(* IEC 61131-3 sources: moqui-plc/simatic-ax/src/moqui/framework/src/main/org/moqui/context, 9 files *)

(* ---- LogCmd.st ---- *)
TYPE LogCmd : (
    Idle, (* Waiting for commands *)
    Push, (* Inserting a new log entry *)
	IncrementLast, (* Update the last log entry *)
	Peek, (* Read a log entry without removing it *)
	Pop, (* It actually removes the appended log entries *)
    Clear (* Complete buffer reset *)
); END_TYPE

(* ---- LogEvent.st ---- *)
TYPE LogEvent : STRUCT
	(* Unique identifier for the log event *)
    logEventId : STRING;
    loggerName : STRING;
	marker : LogMarker;
    level : LogLevel;
    logEventDate : DATE_AND_TIME;
	source : STRING;
	payloadType : LogPayloadType;
    payload : LogPayload;
	(* contextData: STRING; *)
	(* Number of times this log event was repeated, for compression *)
    repeatCount : UINT;
END_STRUCT; END_TYPE

(* ---- LogLevel.st ---- *)
TYPE LogLevel : (
	Trace,
	Debug,
	Info,
	Warn,
	Error,
	Fatal,
	All,
	Off
); END_TYPE

(* ---- LogMarker.st ---- *)
TYPE LogMarker : (
	Diagnostics,
	Lifecycle,
	Integration,
	Health,
	Telemetry,
	AuditLog,
	Kpi,
	Measurement
); END_TYPE

(* ---- LogPayload.st ---- *)
TYPE LogPayload : STRUCT
	message : STRING;
    enumValue : UINT;
    numericValue : LREAL;
END_STRUCT; END_TYPE

(* ---- LogPayloadType.st ---- *)
TYPE LogPayloadType : (
    Text,
	Numeric,
	Enum
); END_TYPE

(* ---- LogSource.st ---- *)
TYPE LogSource : STRUCT
	(* Reference to log ring buffer *)
    logRef : REF_TO LogRingBuffer;
	lastLogSize : UINT;
	lastHead : UINT := UINT#1;
	lastTail : UINT := UINT#1;
	lastOverflowCount : UDINT;
END_STRUCT; END_TYPE

(* ---- LoggerFacade.st ---- *)
(*
 * Logger with local circular buffer and duplicate suppression.
 * Designed for central orchestration by a global LogAppender.
 *)
FUNCTION_BLOCK LoggerFacade
	VAR_EXTERNAL CONSTANT
		defaultLogLevel : LogLevel;
		defaultLogSuppressDuration : TIME;
		defaultLogSuppressDuplicates : BOOL;
		LOG_SOURCE_LIST_MAX_SIZE : UINT;
	END_VAR
	VAR_EXTERNAL
		logSourceList : ARRAY[1..LOG_SOURCE_LIST_MAX_SIZE] OF LogSource;
		logSourceListSize : UINT;
	END_VAR
	(* Log event data *)
	VAR_INPUT
		enable : BOOL;
		logEventId : STRING := '';
		loggerName : STRING;
		level : LogLevel := defaultLogLevel;
		marker : LogMarker := LogMarker#Diagnostics;
		source : STRING;
		payloadType : LogPayloadType := LogPayloadType#Text;
		message : STRING;
		enumValue : UINT;
		numericValue : LREAL;
	END_VAR
	(* Configuration parameters *)
	VAR_INPUT
		suppressDuplicates : BOOL := defaultLogSuppressDuplicates;
		suppressDuration : TIME := defaultLogSuppressDuration;
	END_VAR
	VAR_OUTPUT
		done : BOOL;
		error : BOOL;
	END_VAR
	VAR
		(* Local log ring buffer *)
		logBuffer : LogRingBuffer;
		init : BOOL := FALSE;
		isDuplicate : BOOL;
		now : DATE_AND_TIME;
		lastLogEvent : LogEvent;
		(* Log event ID generator *)
		eventSequence : UDINT := UDINT#0;
	END_VAR

	(* Register once into the log appender source list *)
	IF NOT init THEN
		IF logSourceListSize < LOG_SOURCE_LIST_MAX_SIZE THEN
			logSourceListSize := logSourceListSize + UINT#1;
			logSourceList[logSourceListSize].logRef := REF(logBuffer);
		ELSE
			error := TRUE;
		END_IF;
		init := TRUE;
	END_IF;

	IF NOT enable THEN
		done := FALSE;
		RETURN;
	END_IF;

	now := nowTimestamp();
	isDuplicate := FALSE;

	(* Compression logic (duplicate suppression) *)
	IF suppressDuplicates AND (payloadType = lastLogEvent.payloadType)
			AND (loggerName = lastLogEvent.loggerName)
			AND (source = lastLogEvent.source) THEN
		CASE payloadType OF
			LogPayloadType#Text: isDuplicate := (message = lastLogEvent.payload.message);
			LogPayloadType#Enum: isDuplicate := (enumValue = lastLogEvent.payload.enumValue);
			LogPayloadType#Numeric: isDuplicate := (numericValue = lastLogEvent.payload.numericValue);
		END_CASE;
	END_IF;

	IF isDuplicate AND ((now - lastLogEvent.logEventDate) < suppressDuration) THEN
		(* Increment repeat counter instead of storing new entry *)
		logBuffer.cmd := LogCmd#IncrementLast;
	ELSE
		(* Prepare the new log event entry *)
		IF logEventId = '' THEN
			eventSequence := eventSequence + UDINT#1;
			lastLogEvent.logEventId := loggerName;
		ELSE
			lastLogEvent.logEventId := logEventId;
		END_IF;

		lastLogEvent.loggerName := loggerName;
		lastLogEvent.level := level;
		lastLogEvent.marker := marker;
		lastLogEvent.logEventDate := now;
		lastLogEvent.source := source;
		lastLogEvent.payloadType := payloadType;
		lastLogEvent.repeatCount := UINT#1;

		CASE payloadType OF
			LogPayloadType#Text: lastLogEvent.payload.message := message;
			LogPayloadType#Enum: lastLogEvent.payload.enumValue := enumValue;
			LogPayloadType#Numeric: lastLogEvent.payload.numericValue := numericValue;
		END_CASE;

		(* Append the new log event *)
		logBuffer.logEntry := lastLogEvent;
		logBuffer.cmd := LogCmd#Push;
	END_IF;

	(* Execute local buffer operation *)
	logBuffer();
	logBuffer.cmd := LogCmd#Idle;

	done := logBuffer.done;
	error := error OR logBuffer.error;
END_FUNCTION_BLOCK

(* ---- LogRingBuffer.st ---- *)
FUNCTION_BLOCK LogRingBuffer
	VAR_EXTERNAL CONSTANT
	    LOG_MAX_SIZE : UINT;
	END_VAR
	VAR_INPUT
	    cmd : LogCmd := LogCmd#Idle;
	    logEntry : LogEvent;
	END_VAR
	VAR_OUTPUT
	    done, error, isFull, isEmpty : BOOL;
	    head : UINT := UINT#1;
	    tail : UINT := UINT#1;
	    (* Peek/Pop result: set on LogCmd#Peek and LogCmd#Pop *)
	    headEntry : LogEvent;
	    (* Exposed so that it can be cloned by the log appender (memcpy one-cycle operation). *)
	    logBuffer : ARRAY[1..LOG_MAX_SIZE] OF LogEvent;
	    logSize : UINT;
	    overflowCount : UDINT;
	END_VAR
	VAR CONSTANT
		MAX_UDINT : UDINT := UDINT#16#FFFFFFFF;
	END_VAR
	VAR
	    lastCommand : LogCmd := LogCmd#Idle;
	    i : UINT;
	END_VAR

	(* Reset instant outputs *)
	done := FALSE;
	error := FALSE;

	(* Invariants guard *)
	IF (head < UINT#1) OR (head > LOG_MAX_SIZE) OR (tail < UINT#1) OR (tail > LOG_MAX_SIZE) OR (logSize > LOG_MAX_SIZE) THEN
	    head := UINT#1; tail := UINT#1; logSize := UINT#0;
	    error := TRUE;
	    RETURN;
	END_IF;

	IF (overflowCount = MAX_UDINT) THEN overflowCount := UDINT#1; END_IF;

	IF (cmd <> LogCmd#Idle) THEN
	    CASE cmd OF
	        LogCmd#Push :
	            logBuffer[tail] := logEntry;

	            IF (logSize >= LOG_MAX_SIZE) THEN
	                (* Buffer full, overwrite oldest entries *)
	                head := (head MOD LOG_MAX_SIZE) + UINT#1;
	                overflowCount := overflowCount + UDINT#1;
	            ELSE
	                logSize := logSize + UINT#1;
	            END_IF;

	            tail := (tail MOD LOG_MAX_SIZE) + UINT#1;
	            done := TRUE;

	        (* Increment repeat counter instead of storing new log entry *)
	        LogCmd#IncrementLast :
	            IF logSize = UINT#0 THEN
					error := TRUE;
				ELSE
	                i := tail - UINT#1;
	                IF i < UINT#1 THEN i := LOG_MAX_SIZE; END_IF;

	                (* Saturate repeatCount *)
	                IF logBuffer[i].repeatCount < UINT#65535 THEN
	                    logBuffer[i].repeatCount := logBuffer[i].repeatCount + UINT#1;
	                END_IF;

					done := TRUE;
	            END_IF;

	        (* Returns head entry without removing it. Error if empty (Java Queue.peek semantics). *)
	        LogCmd#Peek :
	            IF logSize = UINT#0 THEN
	                error := TRUE;
	            ELSE
	                headEntry := logBuffer[head];
	                done := TRUE;
	            END_IF;

	        (* Returns and removes head entry. Error if empty (Java Deque.pop semantics). *)
	        LogCmd#Pop :
	            IF logSize = UINT#0 THEN
	                error := TRUE;
	            ELSE
	                headEntry := logBuffer[head];
	                head := (head MOD LOG_MAX_SIZE) + UINT#1;
	                logSize := logSize - UINT#1;
	                done := TRUE;
	            END_IF;

	        LogCmd#Clear :
	            head := UINT#1; tail := UINT#1; logSize := UINT#0; overflowCount := UDINT#0;
	            done := TRUE;
	    END_CASE;
	END_IF;

	lastCommand := cmd;
	isEmpty := (logSize = UINT#0);
	isFull := (logSize = LOG_MAX_SIZE);
	END_FUNCTION_BLOCK
